(* IEC 61131-3 sources: marine-plc-st-examples/, 5 files *)

(* ---- EngineRPM_Calculator.ST ---- *)
PROGRAM EngineRPM_Calculator
VAR
    pulseCount : INT;
    timePeriod : REAL;       // seconds
    RPM        : REAL;
END_VAR

IF timePeriod > 0 THEN
    RPM := (pulseCount / timePeriod) * 60.0; // Convert pulses per second to RPM
END_IF;

(* ---- NMEA_Parser.ST ---- *)
PROGRAM NMEA_Parser
VAR
    sentence  : STRING(100) := '$GPGGA,123519,4807.038,N,01131.000,E';
    lat, lon  : REAL;
END_VAR

// Simple string extraction logic (placeholder)
lat := 48.1173;
lon := 11.5167;

(* ---- PumpControl.ST ---- *)
PROGRAM PumpControl
VAR
    levelLow       : BOOL;      // Low level sensor
    levelHigh      : BOOL;      // High level sensor
    pumpRunning    : BOOL := FALSE;
    manualMode     : BOOL := FALSE;
END_VAR

IF manualMode THEN
    pumpRunning := TRUE; // Manual override
ELSE
    IF levelHigh THEN
        pumpRunning := FALSE; // Stop when tank is full
    ELSIF levelLow THEN
        pumpRunning := TRUE;  // Start when tank is empty
    END_IF;
END_IF;

(* ---- TankFillingSystem.ST ---- *)
PROGRAM TankFillingSystem
VAR
    tankLevel     : REAL;             // Level in %
    highLevel     : REAL := 90.0;     // High-level alarm
    lowLevel      : REAL := 40.0;     // Restart level
    pumpRunning   : BOOL := FALSE;    // Pump output
    highAlarm     : BOOL := FALSE;    // Alarm signal
    manualOverride: BOOL := FALSE;    // Manual mode
END_VAR

IF manualOverride THEN
    // Manual override: Operator forces pump ON
    pumpRunning := TRUE;
    highAlarm := FALSE;
ELSE
    // Automatic control based on tank level
    IF tankLevel >= highLevel THEN
        pumpRunning := FALSE;   // Stop pump when tank is full
        highAlarm := TRUE;      // Trigger alarm
    ELSIF tankLevel <= lowLevel THEN
        pumpRunning := TRUE;    // Restart pump when level is low
        highAlarm := FALSE;
    END_IF;
END_IF;

Add TankFillingSystem structured text example

(* ---- TemperatureAlarm.ST ---- *)
PROGRAM TemperatureAlarm
VAR
    temperature   : REAL;          // Sensor input
    limitHigh     : REAL := 95.0;  // Max allowed
    alarmActive   : BOOL := FALSE;
END_VAR

IF temperature >= limitHigh THEN
    alarmActive := TRUE;
ELSE
    alarmActive := FALSE;
END_IF;
